{attribute 'qualified_only'}
VAR_GLOBAL
	
	bRunning: BOOL;	
	sState :STRING; (*tilatietoa, 80 merkkiä, muutoin string(255) jolloin merkkien pituus 255*)
// yksi merkki on aina yksi byte


END_VAR

(* stored: Version 1.1.0.1, ProductVersion 3.1.4024.0
   GVL VISU: Id {028a7465-f909-40fb-a08e-8c818fe3532d} *)
